// TIA Portal project "babu_2Motors_Simultaneously" (V15)

(* hardware
DEVICE "S7-1200 station_1"  S7-1200 Station
   slot 0: "Rack_0"  S7-1200 Rack  Rack  V1.0
   slot 1: "PLC_1"  CPU 1212C DC/DC/DC  6ES7 212-1AE40-0XB0  V4.2
*)

// ===== PLC "PLC_1"  CPU 1212C DC/DC/DC =====

VAR_GLOBAL   // PLC tag table "Default tag table"
   "PUSH BUTTON 1" AT %M0.0 : Bool;
   "PUSH BUTTON 1 MEMORY" AT %M0.1 : Bool;
   "PUSH BUTTON 2" AT %M0.2 : Bool;
   "PUSH BUTTON 2 MEMORY" AT %M0.3 : Bool;
   "STOP BUTTON" AT %M0.4 : Bool;
   "STOP BUTTON MEMORY" AT %M0.5 : Bool;
   "SIMULATENOUSLY PRESSED" AT %M0.6 : Bool;
   "MOTOR 1" AT %Q0.0 : Bool;
   "MOTOR 2" AT %Q0.1 : Bool;
END_VAR

// folder: System blocks/Program resources

DATA_BLOCK "IEC_Timer_0_DB"   // DB1
{ S7_Optimized_Access := 'TRUE' }
AUTHOR : Simatic
FAMILY : IEC
NAME : IEC_TMR
VERSION : 1.0
// stored: InstanceOfName IEC_TIMER
"IEC_TIMER"
BEGIN
END_DATA_BLOCK

DATA_BLOCK "IEC_Timer_0_DB_1"   // DB2
{ S7_Optimized_Access := 'TRUE' }
AUTHOR : Simatic
FAMILY : IEC
NAME : IEC_TMR
VERSION : 1.0
// stored: InstanceOfName IEC_TIMER
"IEC_TIMER"
BEGIN
END_DATA_BLOCK

DATA_BLOCK "IEC_Timer_0_DB_2"   // DB3
{ S7_Optimized_Access := 'TRUE' }
AUTHOR : Simatic
FAMILY : IEC
NAME : IEC_TMR
VERSION : 1.0
// stored: InstanceOfName IEC_TIMER
"IEC_TIMER"
BEGIN
END_DATA_BLOCK

DATA_BLOCK "IEC_Timer_0_DB_3"   // DB4
{ S7_Optimized_Access := 'TRUE' }
AUTHOR : Simatic
FAMILY : IEC
NAME : IEC_TMR
VERSION : 1.0
// stored: InstanceOfName IEC_TIMER
"IEC_TIMER"
BEGIN
END_DATA_BLOCK

// folder: (top level)

ORGANIZATION_BLOCK "Main"   // OB1, LAD, ProgramCycle
TITLE = "Main Program Sweep (Cycle)"
{ S7_Optimized_Access := 'TRUE' }
VERSION : 0.1
   VAR_INPUT
      Initial_Call : Bool;   // Initial call of this OB
      Remanence : Bool;   // =True, if remanent data are available
   END_VAR
   VAR_TEMP   // added for the SCL form of the ladder/FBD networks
      _w1 : Bool;
      _w2 : Bool;
      _w3 : Bool;
   END_VAR
BEGIN

REGION Network 1
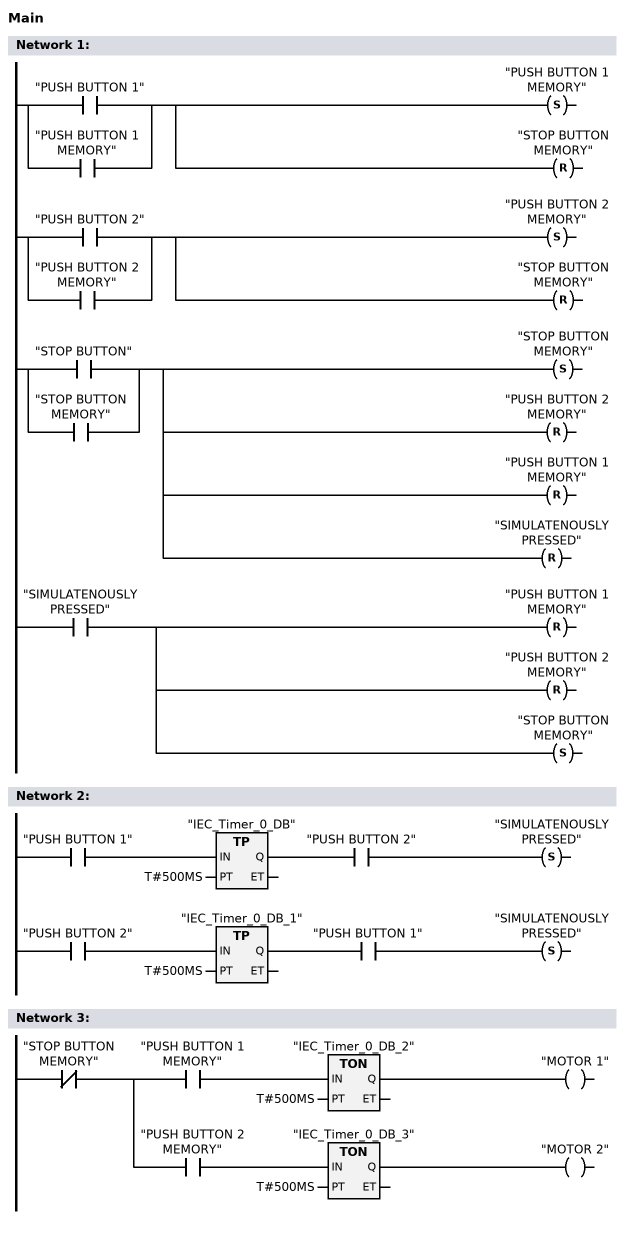
   RUNG wire#powerrail
      Contact( "PUSH BUTTON 1" )
      wire#w1
      S_Coil( "PUSH BUTTON 1 MEMORY" )
   END_RUNG
   RUNG wire#powerrail
      Contact( "PUSH BUTTON 1 MEMORY" )
   END_RUNG wire#w1
   RUNG wire#w1
      R_Coil( "STOP BUTTON MEMORY" )
   END_RUNG
   RUNG wire#powerrail
      Contact( "PUSH BUTTON 2" )
      wire#w2
      S_Coil( "PUSH BUTTON 2 MEMORY" )
   END_RUNG
   RUNG wire#powerrail
      Contact( "PUSH BUTTON 2 MEMORY" )
   END_RUNG wire#w2
   RUNG wire#w2
      R_Coil( "STOP BUTTON MEMORY" )
   END_RUNG
   RUNG wire#powerrail
      Contact( "STOP BUTTON" )
      wire#w3
      S_Coil( "STOP BUTTON MEMORY" )
   END_RUNG
   RUNG wire#powerrail
      Contact( "STOP BUTTON MEMORY" )
   END_RUNG wire#w3
   RUNG wire#w3
      R_Coil( "PUSH BUTTON 2 MEMORY" )
   END_RUNG
   RUNG wire#w3
      R_Coil( "PUSH BUTTON 1 MEMORY" )
   END_RUNG
   RUNG wire#w3
      R_Coil( "SIMULATENOUSLY PRESSED" )
   END_RUNG
   RUNG wire#powerrail
      Contact( "SIMULATENOUSLY PRESSED" )
      wire#w4
      R_Coil( "PUSH BUTTON 1 MEMORY" )
   END_RUNG
   RUNG wire#w4
      R_Coil( "PUSH BUTTON 2 MEMORY" )
   END_RUNG
   RUNG wire#w4
      S_Coil( "STOP BUTTON MEMORY" )
   END_RUNG
   // the same network as SCL:
   #_w1 := "PUSH BUTTON 1" OR "PUSH BUTTON 1 MEMORY";
   IF #_w1 THEN
       "PUSH BUTTON 1 MEMORY" := TRUE;
       "STOP BUTTON MEMORY" := FALSE;
   END_IF;
   #_w2 := "PUSH BUTTON 2" OR "PUSH BUTTON 2 MEMORY";
   IF #_w2 THEN
       "PUSH BUTTON 2 MEMORY" := TRUE;
       "STOP BUTTON MEMORY" := FALSE;
   END_IF;
   #_w3 := "STOP BUTTON" OR "STOP BUTTON MEMORY";
   IF #_w3 THEN
       "STOP BUTTON MEMORY" := TRUE;
       "PUSH BUTTON 2 MEMORY" := FALSE;
       "PUSH BUTTON 1 MEMORY" := FALSE;
       "SIMULATENOUSLY PRESSED" := FALSE;
   END_IF;
   IF "SIMULATENOUSLY PRESSED" THEN
       "PUSH BUTTON 1 MEMORY" := FALSE;
       "PUSH BUTTON 2 MEMORY" := FALSE;
       "STOP BUTTON MEMORY" := TRUE;
   END_IF;
END_REGION

REGION Network 2
   "IEC_Timer_0_DB".TP(IN := "PUSH BUTTON 1", PT := T#500MS);
   IF "IEC_Timer_0_DB".Q AND "PUSH BUTTON 2" THEN "SIMULATENOUSLY PRESSED" := TRUE; END_IF;
   "IEC_Timer_0_DB_1".TP(IN := "PUSH BUTTON 2", PT := T#500MS);
   IF "IEC_Timer_0_DB_1".Q AND "PUSH BUTTON 1" THEN "SIMULATENOUSLY PRESSED" := TRUE; END_IF;
END_REGION

REGION Network 3
   "IEC_Timer_0_DB_2".TON(IN := NOT "STOP BUTTON MEMORY" AND "PUSH BUTTON 1 MEMORY", PT := T#500MS);
   "MOTOR 1" := "IEC_Timer_0_DB_2".Q;
   "IEC_Timer_0_DB_3".TON(IN := NOT "STOP BUTTON MEMORY" AND "PUSH BUTTON 2 MEMORY", PT := T#500MS);
   "MOTOR 2" := "IEC_Timer_0_DB_3".Q;
END_REGION
END_ORGANIZATION_BLOCK